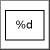
VISUALIZATION diagProfiNetSlave  // 50x50
VAR_IN_OUT
	dataValues:typeProfiNETIndicator;
END_VAR
    Rectangle (0,0 50x50), invisible if: dataValues.SlaveNumber = 0, colour variable: dataValues.historicalState.colour
    Rectangle (5,10 39x30), "%d", text variable: dataValues.SlaveNumber, invisible if: dataValues.SlaveNumber = 0, colour variable: dataValues.currentState.colour
    Rectangle (0,0 50x50), invisible if: dataValues.SlaveNumber = 0
        OnMouseClick: execute { ProfiNetDiag.detailDiagNum := dataValues.SlaveNumber; }
        OnMouseClick: CloseDialog Dialog=diagProfiNetSlaveDetail, Result=OK, NumpadKeypadSet=True
        OnMouseClick: OpenDialog Dialog=diagProfiNetSlaveDetail, OpenModal=True, PositionX=200, PositionY=75
END_VISUALIZATION

(* stored: Version 1.1.0.1, ProductVersion 3.1.4024.12
   Visu diagProfiNetSlave: Id {520379a1-4f71-457d-8f27-6dc6fa557da9} *)
